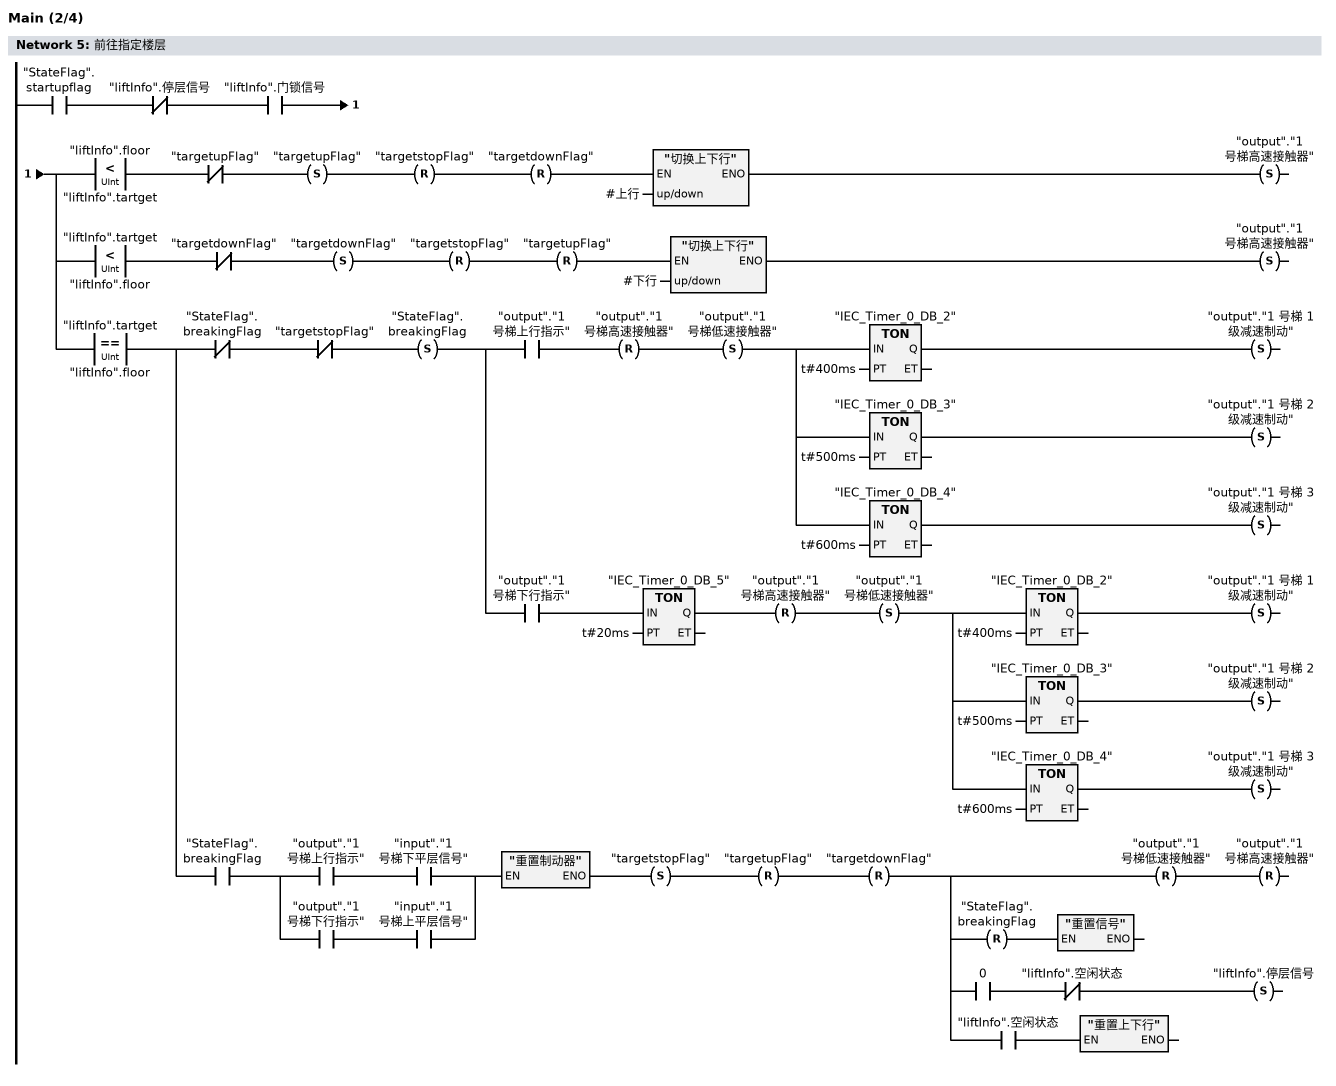
   #_w1 := "StateFlag".startupflag AND NOT "liftInfo".停层信号 AND "liftInfo".门锁信号;
   #_w2 := #_w1 AND ("liftInfo".floor < "liftInfo".tartget) AND NOT "targetupFlag";
   IF #_w2 THEN
       "targetupFlag" := TRUE;
       "targetstopFlag" := FALSE;
       "targetdownFlag" := FALSE;
   END_IF;
   "切换上下行"(EN := #_w2, "up/down" := #上行, ENO => #_w3);
   IF #_w3 THEN "output"."1 号梯高速接触器" := TRUE; END_IF;
   #_w4 := #_w1 AND ("liftInfo".tartget < "liftInfo".floor) AND NOT "targetdownFlag";
   IF #_w4 THEN
       "targetdownFlag" := TRUE;
       "targetstopFlag" := FALSE;
       "targetupFlag" := FALSE;
   END_IF;
   "切换上下行"(EN := #_w4, "up/down" := #下行, ENO => #_w5);
   IF #_w5 THEN "output"."1 号梯高速接触器" := TRUE; END_IF;
   #_w6 := #_w1 AND ("liftInfo".tartget = "liftInfo".floor);
   #_w7 := #_w6 AND NOT "StateFlag".breakingFlag AND NOT "targetstopFlag";
   IF #_w7 THEN "StateFlag".breakingFlag := TRUE; END_IF;
   #_w8 := #_w7 AND "output"."1 号梯上行指示";
   IF #_w8 THEN
       "output"."1 号梯高速接触器" := FALSE;
       "output"."1 号梯低速接触器" := TRUE;
   END_IF;
   "IEC_Timer_0_DB_2".TON(IN := #_w8, PT := t#400ms);
   IF "IEC_Timer_0_DB_2".Q THEN "output"."1 号梯 1 级减速制动" := TRUE; END_IF;
   "IEC_Timer_0_DB_3".TON(IN := #_w8, PT := t#500ms);
   IF "IEC_Timer_0_DB_3".Q THEN "output"."1 号梯 2 级减速制动" := TRUE; END_IF;
   "IEC_Timer_0_DB_4".TON(IN := #_w8, PT := t#600ms);
   IF "IEC_Timer_0_DB_4".Q THEN "output"."1 号梯 3 级减速制动" := TRUE; END_IF;
   "IEC_Timer_0_DB_5".TON(IN := #_w7 AND "output"."1 号梯下行指示", PT := t#20ms);
   IF "IEC_Timer_0_DB_5".Q THEN
       "output"."1 号梯高速接触器" := FALSE;
       "output"."1 号梯低速接触器" := TRUE;
   END_IF;
   "IEC_Timer_0_DB_2".TON(IN := "IEC_Timer_0_DB_5".Q, PT := t#400ms);
   IF "IEC_Timer_0_DB_2".Q THEN "output"."1 号梯 1 级减速制动" := TRUE; END_IF;
   "IEC_Timer_0_DB_3".TON(IN := "IEC_Timer_0_DB_5".Q, PT := t#500ms);
   IF "IEC_Timer_0_DB_3".Q THEN "output"."1 号梯 2 级减速制动" := TRUE; END_IF;
   "IEC_Timer_0_DB_4".TON(IN := "IEC_Timer_0_DB_5".Q, PT := t#600ms);
   IF "IEC_Timer_0_DB_4".Q THEN "output"."1 号梯 3 级减速制动" := TRUE; END_IF;
   "重置制动器"(EN := #_w6 AND "StateFlag".breakingFlag AND (("output"."1 号梯上行指示" AND "input"."1 号梯下平层信号") OR ("output"."1 号梯下行指示" AND "input"."1 号梯上平层信号")),
           ENO => #_w9);
   IF #_w9 THEN
       "targetstopFlag" := TRUE;
       "targetupFlag" := FALSE;
       "targetdownFlag" := FALSE;
       "output"."1 号梯低速接触器" := FALSE;
       "output"."1 号梯高速接触器" := FALSE;
       "StateFlag".breakingFlag := FALSE;
       "重置信号"();
   END_IF;
   IF #_w9 AND 0 AND NOT "liftInfo".空闲状态 THEN "liftInfo".停层信号 := TRUE; END_IF;
   IF #_w9 AND "liftInfo".空闲状态 THEN "重置上下行"(); END_IF;
END_REGION

REGION Network 6: 空闲状态
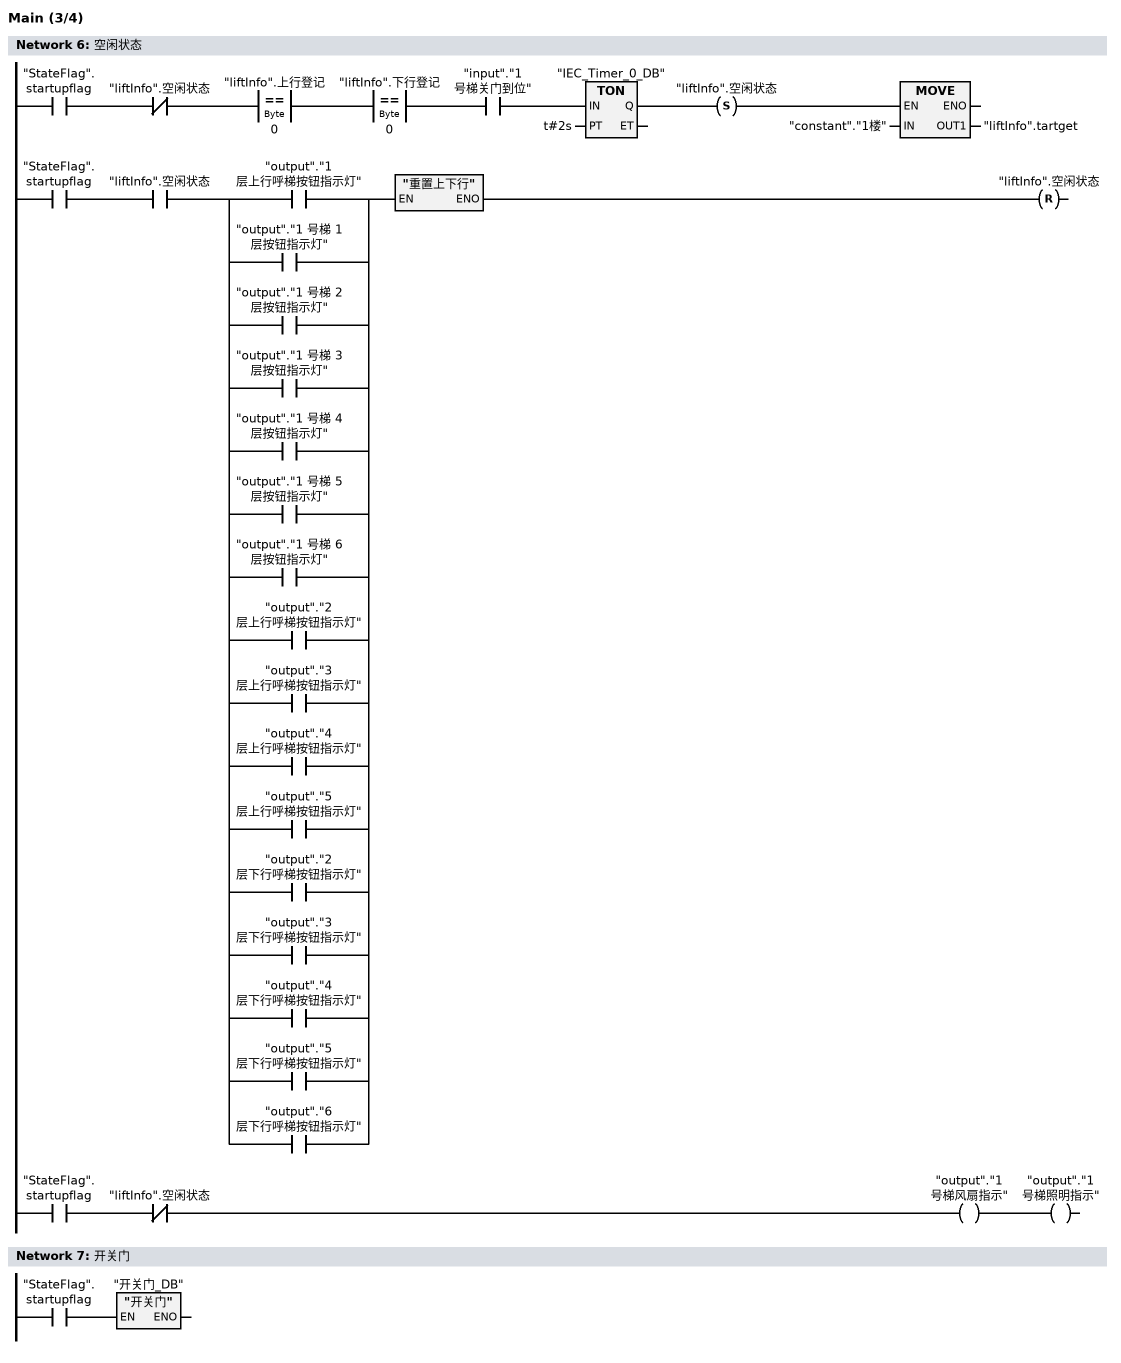
   "IEC_Timer_0_DB".TON(IN := "StateFlag".startupflag AND NOT "liftInfo".空闲状态 AND ("liftInfo".上行登记 = 0) AND ("liftInfo".下行登记 = 0) AND "input"."1 号梯关门到位",
                        PT := t#2s);
   IF "IEC_Timer_0_DB".Q THEN
       "liftInfo".空闲状态 := TRUE;
       "liftInfo".tartget := "constant"."1楼";
   END_IF;
   "重置上下行"(EN := "StateFlag".startupflag AND "liftInfo".空闲状态 AND ("output"."1 层上行呼梯按钮指示灯" OR "output"."1 号梯 1 层按钮指示灯" OR "output"."1 号梯 2 层按钮指示灯" OR "output"."1 号梯 3 层按钮指示灯" OR "output"."1 号梯 4 层按钮指示灯" OR "output"."1 号梯 5 层按钮指示灯" OR "output"."1 号梯 6 层按钮指示灯" OR "output"."2 层上行呼梯按钮指示灯" OR "output"."3 层上行呼梯按钮指示灯" OR "output"."4 层上行呼梯按钮指示灯" OR "output"."5 层上行呼梯按钮指示灯" OR "output"."2 层下行呼梯按钮指示灯" OR "output"."3 层下行呼梯按钮指示灯" OR "output"."4 层下行呼梯按钮指示灯" OR "output"."5 层下行呼梯按钮指示灯" OR "output"."6 层下行呼梯按钮指示灯"),
           ENO => #_w1);
   IF #_w1 THEN "liftInfo".空闲状态 := FALSE; END_IF;
   "output"."1 号梯风扇指示" := "StateFlag".startupflag AND NOT "liftInfo".空闲状态;
   "output"."1 号梯照明指示" := "output"."1 号梯风扇指示";
END_REGION

REGION Network 7: 开关门
   RUNG wire#powerrail
      Contact( "StateFlag".startupflag )
      "开关门_DB"()
   END_RUNG
   // the same network as SCL:
   IF "StateFlag".startupflag THEN
       "开关门_DB"();   // "开关门"
   END_IF;
END_REGION

REGION Network 8: 自动关门
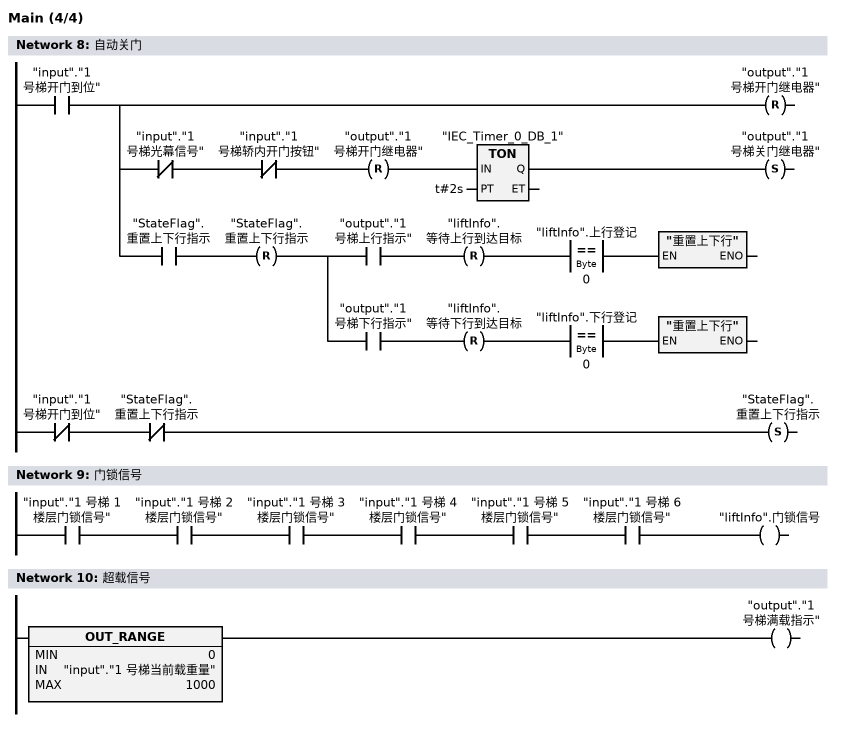
   IF "input"."1 号梯开门到位" THEN "output"."1 号梯开门继电器" := FALSE; END_IF;
   #_w1 := "input"."1 号梯开门到位" AND NOT "input"."1 号梯光幕信号" AND NOT "input"."1 号梯轿内开门按钮";
   IF #_w1 THEN "output"."1 号梯开门继电器" := FALSE; END_IF;
   "IEC_Timer_0_DB_1".TON(IN := #_w1, PT := t#2s);
   IF "IEC_Timer_0_DB_1".Q THEN "output"."1 号梯关门继电器" := TRUE; END_IF;
   #_w2 := "input"."1 号梯开门到位" AND "StateFlag".重置上下行指示;
   IF #_w2 THEN "StateFlag".重置上下行指示 := FALSE; END_IF;
   #_w3 := #_w2 AND "output"."1 号梯上行指示";
   IF #_w3 THEN "liftInfo".等待上行到达目标 := FALSE; END_IF;
   IF #_w3 AND ("liftInfo".上行登记 = 0) THEN "重置上下行"(); END_IF;
   #_w4 := #_w2 AND "output"."1 号梯下行指示";
   IF #_w4 THEN "liftInfo".等待下行到达目标 := FALSE; END_IF;
   IF #_w4 AND ("liftInfo".下行登记 = 0) THEN "重置上下行"(); END_IF;
   IF NOT "input"."1 号梯开门到位" AND NOT "StateFlag".重置上下行指示 THEN "StateFlag".重置上下行指示 := TRUE; END_IF;
END_REGION

REGION Network 9: 门锁信号
   RUNG wire#powerrail
      Contact( "input"."1 号梯 1 楼层门锁信号" )
      Contact( "input"."1 号梯 2 楼层门锁信号" )
      Contact( "input"."1 号梯 3 楼层门锁信号" )
      Contact( "input"."1 号梯 4 楼层门锁信号" )
      Contact( "input"."1 号梯 5 楼层门锁信号" )
      Contact( "input"."1 号梯 6 楼层门锁信号" )
      Coil( "liftInfo".门锁信号 )
   END_RUNG
   // the same network as SCL:
   "liftInfo".门锁信号 := "input"."1 号梯 1 楼层门锁信号" AND "input"."1 号梯 2 楼层门锁信号" AND "input"."1 号梯 3 楼层门锁信号" AND "input"."1 号梯 4 楼层门锁信号" AND "input"."1 号梯 5 楼层门锁信号" AND "input"."1 号梯 6 楼层门锁信号";
END_REGION

REGION Network 10: 超载信号
   "output"."1 号梯满载指示" := ("input"."1 号梯当前载重量" < 0) OR ("input"."1 号梯当前载重量" > 1000);
END_REGION
END_ORGANIZATION_BLOCK

ORGANIZATION_BLOCK "Initialize"   // OB124, LAD, ProgramCycle
TITLE = "Main Program Sweep (Cycle)"
{ S7_Optimized_Access := 'TRUE' }
VERSION : 0.1
   VAR_INPUT
      Initial_Call : Bool;   // Initial call of this OB
      Remanence : Bool;   // =True, if remanent data are available
   END_VAR
   VAR_TEMP   // added for the SCL form of the ladder/FBD networks
      _w1 : Bool;
      _w2 : Bool;
      _w3 : Bool;
      _w4 : Bool;
      _w5 : Bool;
      _w6 : Bool;
   END_VAR
BEGIN

REGION Network 1: startup
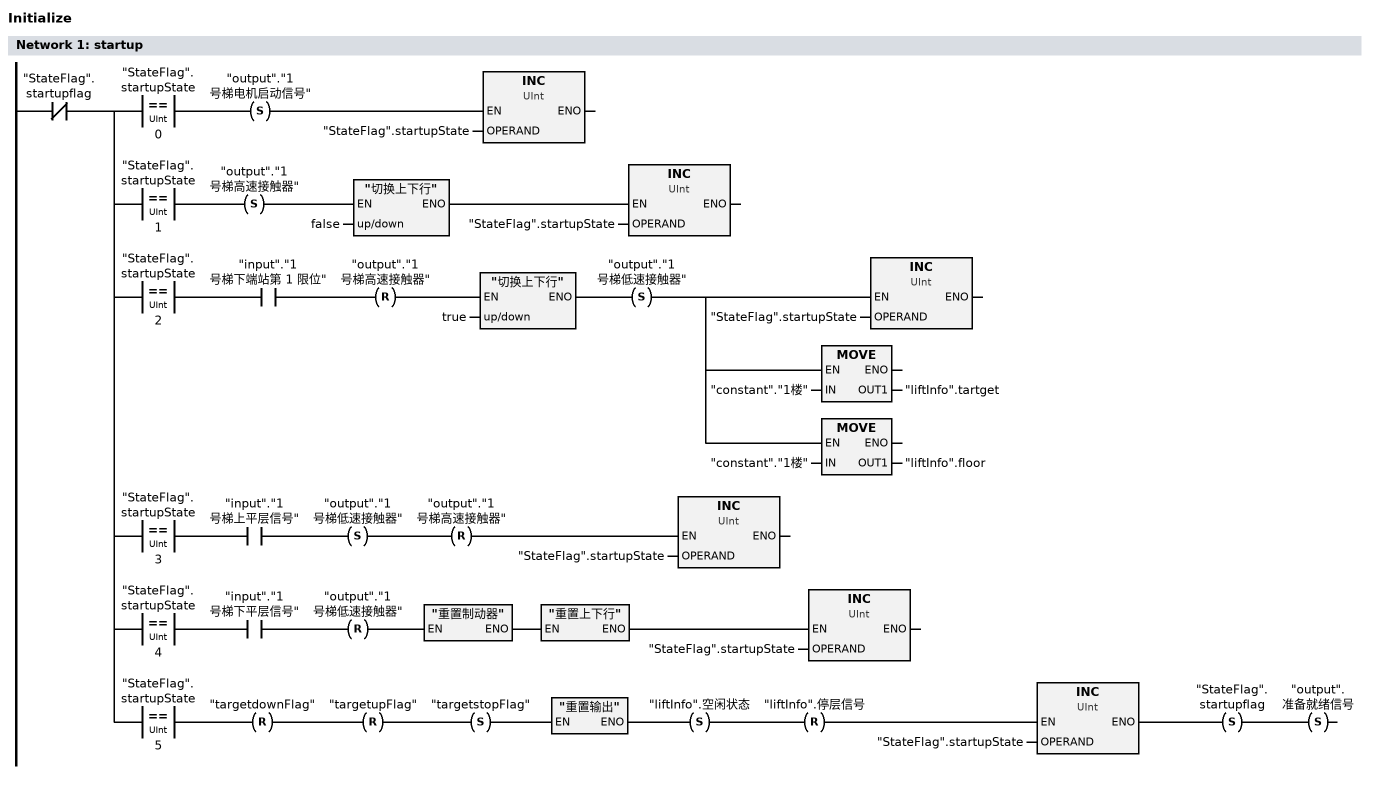
   RUNG wire#powerrail
      I_Contact( "StateFlag".startupflag )
      wire#w1
      { S7_Templates := "SrcType := UInt" } EQ_Contact(in1 := "StateFlag".startupState, in2 := 0)
      S_Coil( "output"."1 号梯电机启动信号" )
      { S7_Templates := "DestType := UInt" } Inc( "StateFlag".startupState )
   END_RUNG
   RUNG wire#w1
      { S7_Templates := "SrcType := UInt" } EQ_Contact(in1 := "StateFlag".startupState, in2 := 1)
      S_Coil( "output"."1 号梯高速接触器" )
      "切换上下行"("up/down" := false)
      { S7_Templates := "DestType := UInt" } Inc( "StateFlag".startupState )
   END_RUNG
   RUNG wire#w1
      { S7_Templates := "SrcType := UInt" } EQ_Contact(in1 := "StateFlag".startupState, in2 := 2)
      Contact( "input"."1 号梯下端站第 1 限位" )
      R_Coil( "output"."1 号梯高速接触器" )
      "切换上下行"("up/down" := true)
      S_Coil( "output"."1 号梯低速接触器" )
      wire#w2
      { S7_Templates := "DestType := UInt" } Inc( "StateFlag".startupState )
   END_RUNG
   RUNG wire#w2
      Move(in := "constant"."1楼", out1 => "liftInfo".tartget)
   END_RUNG
   RUNG wire#w2
      Move(in := "constant"."1楼", out1 => "liftInfo".floor)
   END_RUNG
   RUNG wire#w1
      { S7_Templates := "SrcType := UInt" } EQ_Contact(in1 := "StateFlag".startupState, in2 := 3)
      Contact( "input"."1 号梯上平层信号" )
      S_Coil( "output"."1 号梯低速接触器" )
      R_Coil( "output"."1 号梯高速接触器" )
      { S7_Templates := "DestType := UInt" } Inc( "StateFlag".startupState )
   END_RUNG
   RUNG wire#w1
      { S7_Templates := "SrcType := UInt" } EQ_Contact(in1 := "StateFlag".startupState, in2 := 4)
      Contact( "input"."1 号梯下平层信号" )
      R_Coil( "output"."1 号梯低速接触器" )
      "重置制动器"()
      "重置上下行"()
      { S7_Templates := "DestType := UInt" } Inc( "StateFlag".startupState )
   END_RUNG
   RUNG wire#w1
      { S7_Templates := "SrcType := UInt" } EQ_Contact(in1 := "StateFlag".startupState, in2 := 5)
      R_Coil( "targetdownFlag" )
      R_Coil( "targetupFlag" )
      S_Coil( "targetstopFlag" )
      "重置输出"()
      S_Coil( "liftInfo".空闲状态 )
      R_Coil( "liftInfo".停层信号 )
      { S7_Templates := "DestType := UInt" } Inc( "StateFlag".startupState )
      S_Coil( "StateFlag".startupflag )
      S_Coil( "output".准备就绪信号 )
   END_RUNG
   // the same network as SCL:
   #_w1 := NOT "StateFlag".startupflag;
   IF #_w1 AND ("StateFlag".startupState = 0) THEN
       "output"."1 号梯电机启动信号" := TRUE;
       "StateFlag".startupState := "StateFlag".startupState + 1;
   END_IF;
   IF #_w1 AND ("StateFlag".startupState = 1) THEN "output"."1 号梯高速接触器" := TRUE; END_IF;
   "切换上下行"(EN := #_w1 AND ("StateFlag".startupState = 1), "up/down" := false, ENO => #_w2);
   IF #_w2 THEN "StateFlag".startupState := "StateFlag".startupState + 1; END_IF;
   IF #_w1 AND ("StateFlag".startupState = 2) AND "input"."1 号梯下端站第 1 限位" THEN
       "output"."1 号梯高速接触器" := FALSE;
   END_IF;
   "切换上下行"(EN := #_w1 AND ("StateFlag".startupState = 2) AND "input"."1 号梯下端站第 1 限位",
           "up/down" := true,
           ENO => #_w3);
   IF #_w3 THEN
       "output"."1 号梯低速接触器" := TRUE;
       "StateFlag".startupState := "StateFlag".startupState + 1;
       "liftInfo".tartget := "constant"."1楼";
       "liftInfo".floor := "constant"."1楼";
   END_IF;
   IF #_w1 AND ("StateFlag".startupState = 3) AND "input"."1 号梯上平层信号" THEN
       "output"."1 号梯低速接触器" := TRUE;
       "output"."1 号梯高速接触器" := FALSE;
       "StateFlag".startupState := "StateFlag".startupState + 1;
   END_IF;
   IF #_w1 AND ("StateFlag".startupState = 4) AND "input"."1 号梯下平层信号" THEN
       "output"."1 号梯低速接触器" := FALSE;
   END_IF;
   "重置制动器"(EN := #_w1 AND ("StateFlag".startupState = 4) AND "input"."1 号梯下平层信号", ENO => #_w4);
   "重置上下行"(EN := #_w4, ENO => #_w5);
   IF #_w5 THEN "StateFlag".startupState := "StateFlag".startupState + 1; END_IF;
   IF #_w1 AND ("StateFlag".startupState = 5) THEN
       "targetdownFlag" := FALSE;
       "targetupFlag" := FALSE;
       "targetstopFlag" := TRUE;
   END_IF;
   "重置输出"(EN := #_w1 AND ("StateFlag".startupState = 5), ENO => #_w6);
   IF #_w6 THEN
       "liftInfo".空闲状态 := TRUE;
       "liftInfo".停层信号 := FALSE;
       "StateFlag".startupState := "StateFlag".startupState + 1;
       "StateFlag".startupflag := TRUE;
       "output".准备就绪信号 := TRUE;
   END_IF;
END_REGION
END_ORGANIZATION_BLOCK

ORGANIZATION_BLOCK "外部信号处理"   // OB125, LAD, ProgramCycle
TITLE = "Main Program Sweep (Cycle)"
{ S7_Optimized_Access := 'TRUE' }
VERSION : 0.1
   VAR_INPUT
      Initial_Call : Bool;   // Initial call of this OB
      Remanence : Bool;   // =True, if remanent data are available
   END_VAR
   VAR_TEMP
      tmp1 : Byte;
   END_VAR
   VAR_TEMP   // added for the SCL form of the ladder/FBD networks
      _w1 : Bool;
      _w2 : Bool;
      _w3 : Bool;
      _w4 : Bool;
   END_VAR
BEGIN

REGION Network 1: 处理梯内层按钮
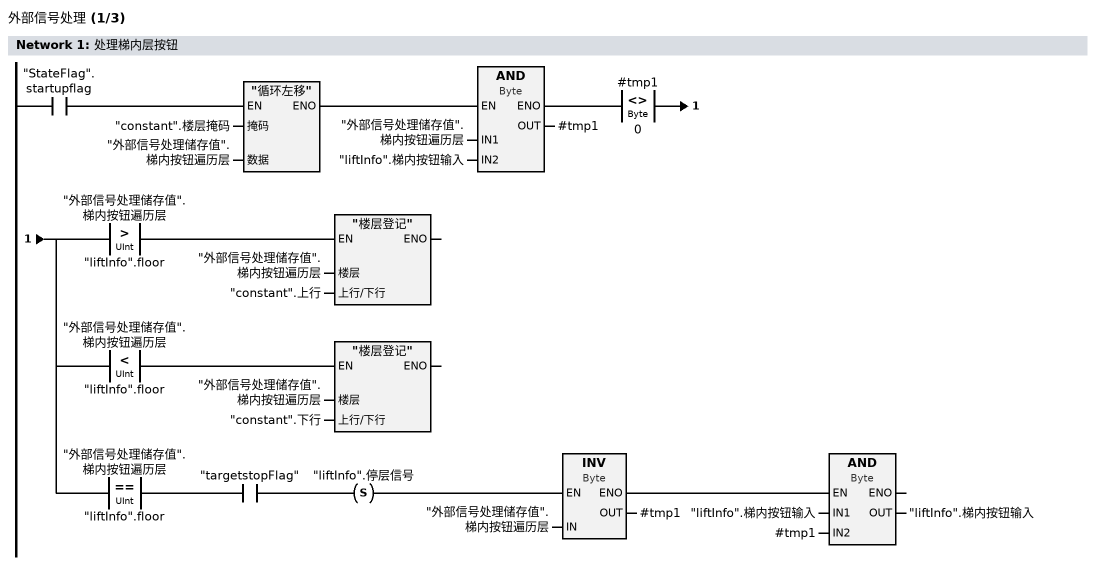
   RUNG wire#powerrail
      Contact( "StateFlag".startupflag )
      "循环左移"(掩码 := "constant".楼层掩码, 数据 := "外部信号处理储存值".梯内按钮遍历层)
      { S7_Templates := "SrcType := Byte" } And(in1 := "外部信号处理储存值".梯内按钮遍历层, in2 := "liftInfo".梯内按钮输入, out => #tmp1)
      { S7_Templates := "SrcType := Byte" } NE_Contact(in1 := #tmp1, in2 := 0)
      wire#w1
      { S7_Templates := "SrcType := UInt" } GT_Contact(in1 := "外部信号处理储存值".梯内按钮遍历层, in2 := "liftInfo".floor)
      "楼层登记"(楼层 := "外部信号处理储存值".梯内按钮遍历层, "上行/下行" := "constant".上行)
   END_RUNG
   RUNG wire#w1
      { S7_Templates := "SrcType := UInt" } LT_Contact(in1 := "外部信号处理储存值".梯内按钮遍历层, in2 := "liftInfo".floor)
      "楼层登记"(楼层 := "外部信号处理储存值".梯内按钮遍历层, "上行/下行" := "constant".下行)
   END_RUNG
   RUNG wire#w1
      { S7_Templates := "SrcType := UInt" } EQ_Contact(in1 := "外部信号处理储存值".梯内按钮遍历层, in2 := "liftInfo".floor)
      Contact( "targetstopFlag" )
      S_Coil( "liftInfo".停层信号 )
      { S7_Templates := "SrcType := Byte" } Inv(in := "外部信号处理储存值".梯内按钮遍历层, out => #tmp1)
      { S7_Templates := "SrcType := Byte" } And(in1 := "liftInfo".梯内按钮输入, in2 := #tmp1, out => "liftInfo".梯内按钮输入)
   END_RUNG
   // the same network as SCL:
   "循环左移"(EN := "StateFlag".startupflag, 掩码 := "constant".楼层掩码, 数据 := "外部信号处理储存值".梯内按钮遍历层, ENO => #_w1);
   IF #_w1 THEN #tmp1 := "外部信号处理储存值".梯内按钮遍历层 AND "liftInfo".梯内按钮输入; END_IF;
   #_w2 := #_w1 AND (#tmp1 <> 0);
   IF #_w2 AND ("外部信号处理储存值".梯内按钮遍历层 > "liftInfo".floor) THEN
       "楼层登记"(楼层 := "外部信号处理储存值".梯内按钮遍历层, "上行/下行" := "constant".上行);
   END_IF;
   IF #_w2 AND ("外部信号处理储存值".梯内按钮遍历层 < "liftInfo".floor) THEN
       "楼层登记"(楼层 := "外部信号处理储存值".梯内按钮遍历层, "上行/下行" := "constant".下行);
   END_IF;
   IF #_w2 AND ("外部信号处理储存值".梯内按钮遍历层 = "liftInfo".floor) AND "targetstopFlag" THEN
       "liftInfo".停层信号 := TRUE;
       #tmp1 := NOT "外部信号处理储存值".梯内按钮遍历层;
       "liftInfo".梯内按钮输入 := "liftInfo".梯内按钮输入 AND #tmp1;
   END_IF;
END_REGION

REGION Network 2: 上行按钮处理
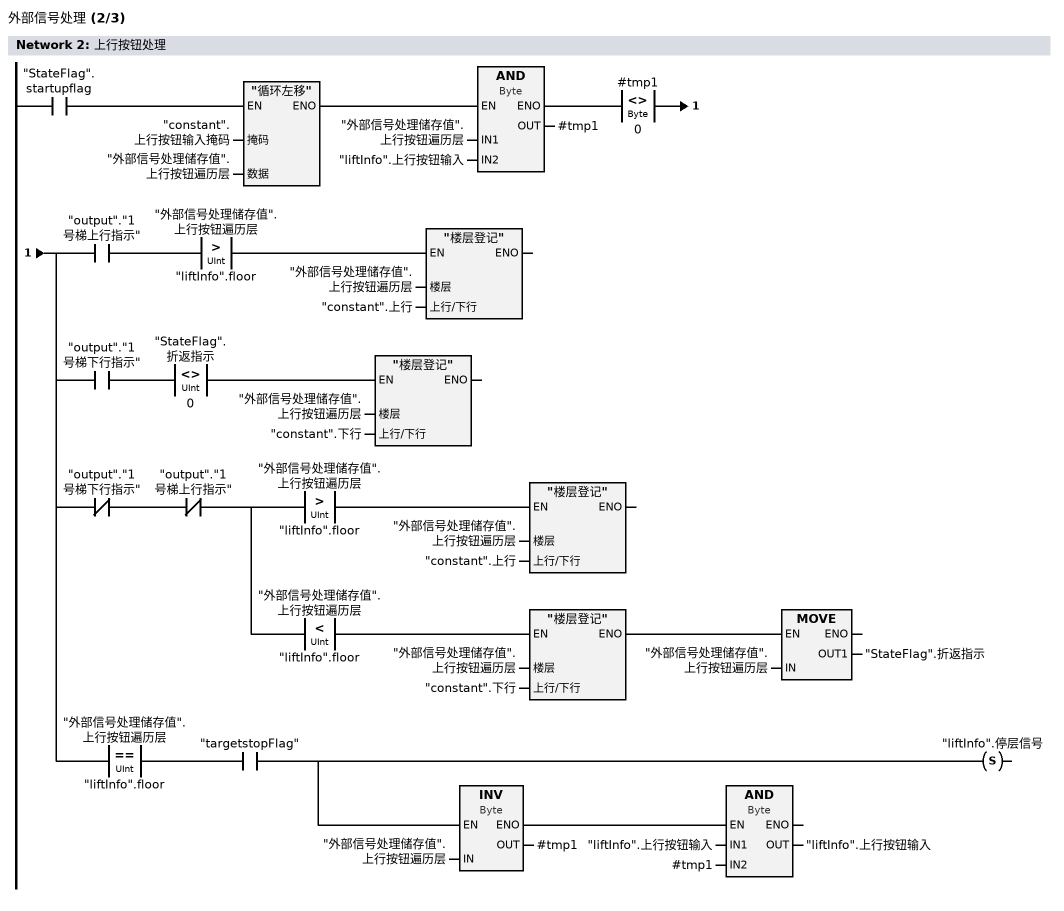
   RUNG wire#powerrail
      Contact( "StateFlag".startupflag )
      "循环左移"(掩码 := "constant".上行按钮输入掩码, 数据 := "外部信号处理储存值".上行按钮遍历层)
      { S7_Templates := "SrcType := Byte" } And(in1 := "外部信号处理储存值".上行按钮遍历层, in2 := "liftInfo".上行按钮输入, out => #tmp1)
      { S7_Templates := "SrcType := Byte" } NE_Contact(in1 := #tmp1, in2 := 0)
      wire#w1
      Contact( "output"."1 号梯上行指示" )
      { S7_Templates := "SrcType := UInt" } GT_Contact(in1 := "外部信号处理储存值".上行按钮遍历层, in2 := "liftInfo".floor)
      "楼层登记"(楼层 := "外部信号处理储存值".上行按钮遍历层, "上行/下行" := "constant".上行)
   END_RUNG
   RUNG wire#w1
      Contact( "output"."1 号梯下行指示" )
      { S7_Templates := "SrcType := UInt" } NE_Contact(in1 := "StateFlag".折返指示, in2 := 0)
      "楼层登记"(楼层 := "外部信号处理储存值".上行按钮遍历层, "上行/下行" := "constant".下行)
   END_RUNG
   RUNG wire#w1
      I_Contact( "output"."1 号梯下行指示" )
      I_Contact( "output"."1 号梯上行指示" )
      wire#w2
      { S7_Templates := "SrcType := UInt" } GT_Contact(in1 := "外部信号处理储存值".上行按钮遍历层, in2 := "liftInfo".floor)
      "楼层登记"(楼层 := "外部信号处理储存值".上行按钮遍历层, "上行/下行" := "constant".上行)
   END_RUNG
   RUNG wire#w2
      { S7_Templates := "SrcType := UInt" } LT_Contact(in1 := "外部信号处理储存值".上行按钮遍历层, in2 := "liftInfo".floor)
      "楼层登记"(楼层 := "外部信号处理储存值".上行按钮遍历层, "上行/下行" := "constant".下行)
      Move(in := "外部信号处理储存值".上行按钮遍历层, out1 => "StateFlag".折返指示)
   END_RUNG
   RUNG wire#w1
      { S7_Templates := "SrcType := UInt" } EQ_Contact(in1 := "外部信号处理储存值".上行按钮遍历层, in2 := "liftInfo".floor)
      Contact( "targetstopFlag" )
      wire#w3
      S_Coil( "liftInfo".停层信号 )
   END_RUNG
   RUNG wire#w3
      { S7_Templates := "SrcType := Byte" } Inv(in := "外部信号处理储存值".上行按钮遍历层, out => #tmp1)
      { S7_Templates := "SrcType := Byte" } And(in1 := "liftInfo".上行按钮输入, in2 := #tmp1, out => "liftInfo".上行按钮输入)
   END_RUNG
   // the same network as SCL:
   "循环左移"(EN := "StateFlag".startupflag, 掩码 := "constant".上行按钮输入掩码, 数据 := "外部信号处理储存值".上行按钮遍历层, ENO => #_w1);
   IF #_w1 THEN #tmp1 := "外部信号处理储存值".上行按钮遍历层 AND "liftInfo".上行按钮输入; END_IF;
   #_w2 := #_w1 AND (#tmp1 <> 0);
   IF #_w2 AND "output"."1 号梯上行指示" AND ("外部信号处理储存值".上行按钮遍历层 > "liftInfo".floor) THEN
       "楼层登记"(楼层 := "外部信号处理储存值".上行按钮遍历层, "上行/下行" := "constant".上行);
   END_IF;
   IF #_w2 AND "output"."1 号梯下行指示" AND ("StateFlag".折返指示 <> 0) THEN
       "楼层登记"(楼层 := "外部信号处理储存值".上行按钮遍历层, "上行/下行" := "constant".下行);
   END_IF;
   #_w3 := #_w2 AND NOT "output"."1 号梯下行指示" AND NOT "output"."1 号梯上行指示";
   IF #_w3 AND ("外部信号处理储存值".上行按钮遍历层 > "liftInfo".floor) THEN
       "楼层登记"(楼层 := "外部信号处理储存值".上行按钮遍历层, "上行/下行" := "constant".上行);
   END_IF;
   "楼层登记"(EN := #_w3 AND ("外部信号处理储存值".上行按钮遍历层 < "liftInfo".floor),
          楼层 := "外部信号处理储存值".上行按钮遍历层,
          "上行/下行" := "constant".下行,
          ENO => #_w4);
   IF #_w4 THEN "StateFlag".折返指示 := "外部信号处理储存值".上行按钮遍历层; END_IF;
   IF #_w2 AND ("外部信号处理储存值".上行按钮遍历层 = "liftInfo".floor) AND "targetstopFlag" THEN
       "liftInfo".停层信号 := TRUE;
       #tmp1 := NOT "外部信号处理储存值".上行按钮遍历层;
       "liftInfo".上行按钮输入 := "liftInfo".上行按钮输入 AND #tmp1;
   END_IF;
END_REGION

REGION Network 3: 下行按钮处理
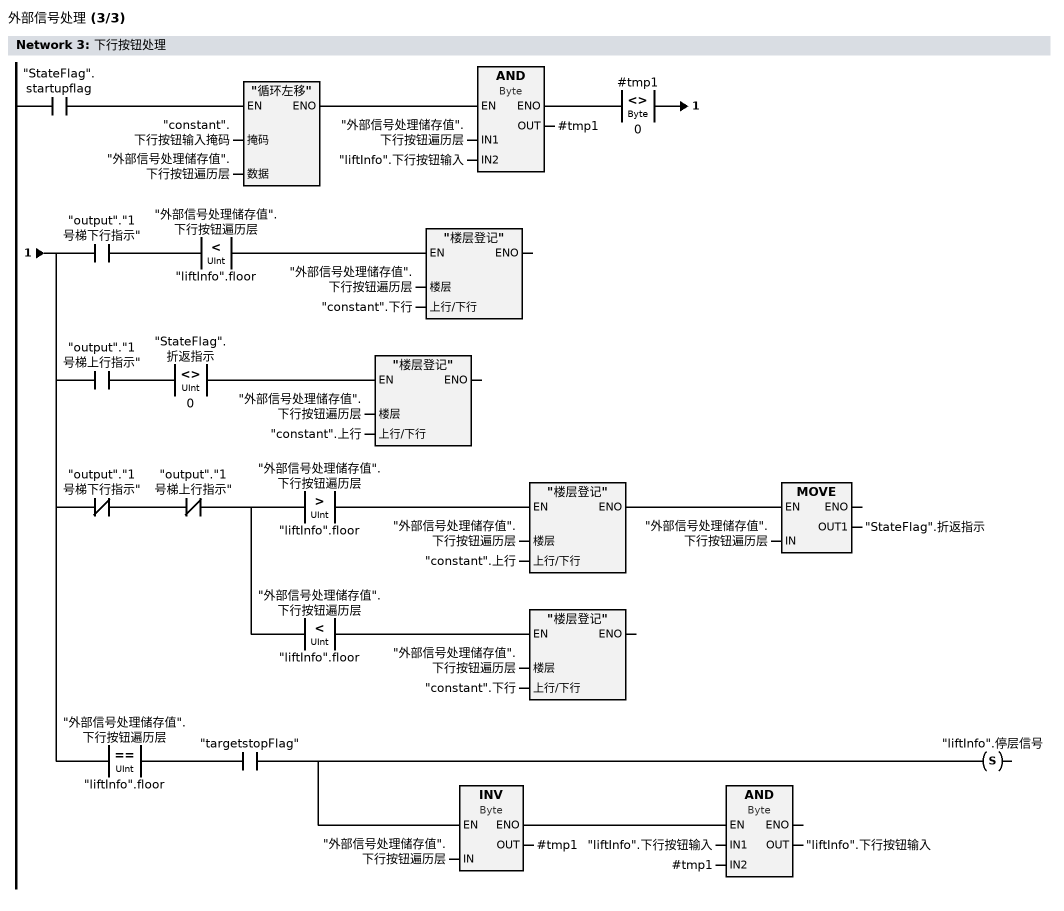
   RUNG wire#powerrail
      Contact( "StateFlag".startupflag )
      "循环左移"(掩码 := "constant".下行按钮输入掩码, 数据 := "外部信号处理储存值".下行按钮遍历层)
      { S7_Templates := "SrcType := Byte" } And(in1 := "外部信号处理储存值".下行按钮遍历层, in2 := "liftInfo".下行按钮输入, out => #tmp1)
      { S7_Templates := "SrcType := Byte" } NE_Contact(in1 := #tmp1, in2 := 0)
      wire#w1
      Contact( "output"."1 号梯下行指示" )
      { S7_Templates := "SrcType := UInt" } LT_Contact(in1 := "外部信号处理储存值".下行按钮遍历层, in2 := "liftInfo".floor)
      "楼层登记"(楼层 := "外部信号处理储存值".下行按钮遍历层, "上行/下行" := "constant".下行)
   END_RUNG
   RUNG wire#w1
      Contact( "output"."1 号梯上行指示" )
      { S7_Templates := "SrcType := UInt" } NE_Contact(in1 := "StateFlag".折返指示, in2 := 0)
      "楼层登记"(楼层 := "外部信号处理储存值".下行按钮遍历层, "上行/下行" := "constant".上行)
   END_RUNG
   RUNG wire#w1
      I_Contact( "output"."1 号梯下行指示" )
      I_Contact( "output"."1 号梯上行指示" )
      wire#w2
      { S7_Templates := "SrcType := UInt" } GT_Contact(in1 := "外部信号处理储存值".下行按钮遍历层, in2 := "liftInfo".floor)
      "楼层登记"(楼层 := "外部信号处理储存值".下行按钮遍历层, "上行/下行" := "constant".上行)
      Move(in := "外部信号处理储存值".下行按钮遍历层, out1 => "StateFlag".折返指示)
   END_RUNG
   RUNG wire#w2
      { S7_Templates := "SrcType := UInt" } LT_Contact(in1 := "外部信号处理储存值".下行按钮遍历层, in2 := "liftInfo".floor)
      "楼层登记"(楼层 := "外部信号处理储存值".下行按钮遍历层, "上行/下行" := "constant".下行)
   END_RUNG
   RUNG wire#w1
      { S7_Templates := "SrcType := UInt" } EQ_Contact(in1 := "外部信号处理储存值".下行按钮遍历层, in2 := "liftInfo".floor)
      Contact( "targetstopFlag" )
      wire#w3
      S_Coil( "liftInfo".停层信号 )
   END_RUNG
   RUNG wire#w3
      { S7_Templates := "SrcType := Byte" } Inv(in := "外部信号处理储存值".下行按钮遍历层, out => #tmp1)
      { S7_Templates := "SrcType := Byte" } And(in1 := "liftInfo".下行按钮输入, in2 := #tmp1, out => "liftInfo".下行按钮输入)
   END_RUNG
   // the same network as SCL:
   "循环左移"(EN := "StateFlag".startupflag, 掩码 := "constant".下行按钮输入掩码, 数据 := "外部信号处理储存值".下行按钮遍历层, ENO => #_w1);
   IF #_w1 THEN #tmp1 := "外部信号处理储存值".下行按钮遍历层 AND "liftInfo".下行按钮输入; END_IF;
   #_w2 := #_w1 AND (#tmp1 <> 0);
   IF #_w2 AND "output"."1 号梯下行指示" AND ("外部信号处理储存值".下行按钮遍历层 < "liftInfo".floor) THEN
       "楼层登记"(楼层 := "外部信号处理储存值".下行按钮遍历层, "上行/下行" := "constant".下行);
   END_IF;
   IF #_w2 AND "output"."1 号梯上行指示" AND ("StateFlag".折返指示 <> 0) THEN
       "楼层登记"(楼层 := "外部信号处理储存值".下行按钮遍历层, "上行/下行" := "constant".上行);
   END_IF;
   #_w3 := #_w2 AND NOT "output"."1 号梯下行指示" AND NOT "output"."1 号梯上行指示";
   "楼层登记"(EN := #_w3 AND ("外部信号处理储存值".下行按钮遍历层 > "liftInfo".floor),
          楼层 := "外部信号处理储存值".下行按钮遍历层,
          "上行/下行" := "constant".上行,
          ENO => #_w4);
   IF #_w4 THEN "StateFlag".折返指示 := "外部信号处理储存值".下行按钮遍历层; END_IF;
   IF #_w3 AND ("外部信号处理储存值".下行按钮遍历层 < "liftInfo".floor) THEN
       "楼层登记"(楼层 := "外部信号处理储存值".下行按钮遍历层, "上行/下行" := "constant".下行);
   END_IF;
   IF #_w2 AND ("外部信号处理储存值".下行按钮遍历层 = "liftInfo".floor) AND "targetstopFlag" THEN
       "liftInfo".停层信号 := TRUE;
       #tmp1 := NOT "外部信号处理储存值".下行按钮遍历层;
       "liftInfo".下行按钮输入 := "liftInfo".下行按钮输入 AND #tmp1;
   END_IF;
END_REGION
END_ORGANIZATION_BLOCK